SYSTEM BaggageSystemCTL (* System Configuration *)
  (* Standard: 61499-1 *)
  (* Version 0.3, 2003-12-05, JHC, Rockwell Automation, Renamed from NEWSYSTEM. *)
  (* Version 0.2, 2002-11-05, JHC, Rockwell Automation, Fixed missing (empty) FBD in Application. *)
  (* Version 0.1, 2002-01-17, JHC, Rockwell Automation, Minor cleanup *)
  (* Version 0.0, 2000-05-27, JHC, Rockwell Automation *)
  APPLICATION APP1
  END_APPLICATION
  DEVICE VIEW : ImageDev(Length := 820, Height := 900)
    RESOURCE RES : ImageResource
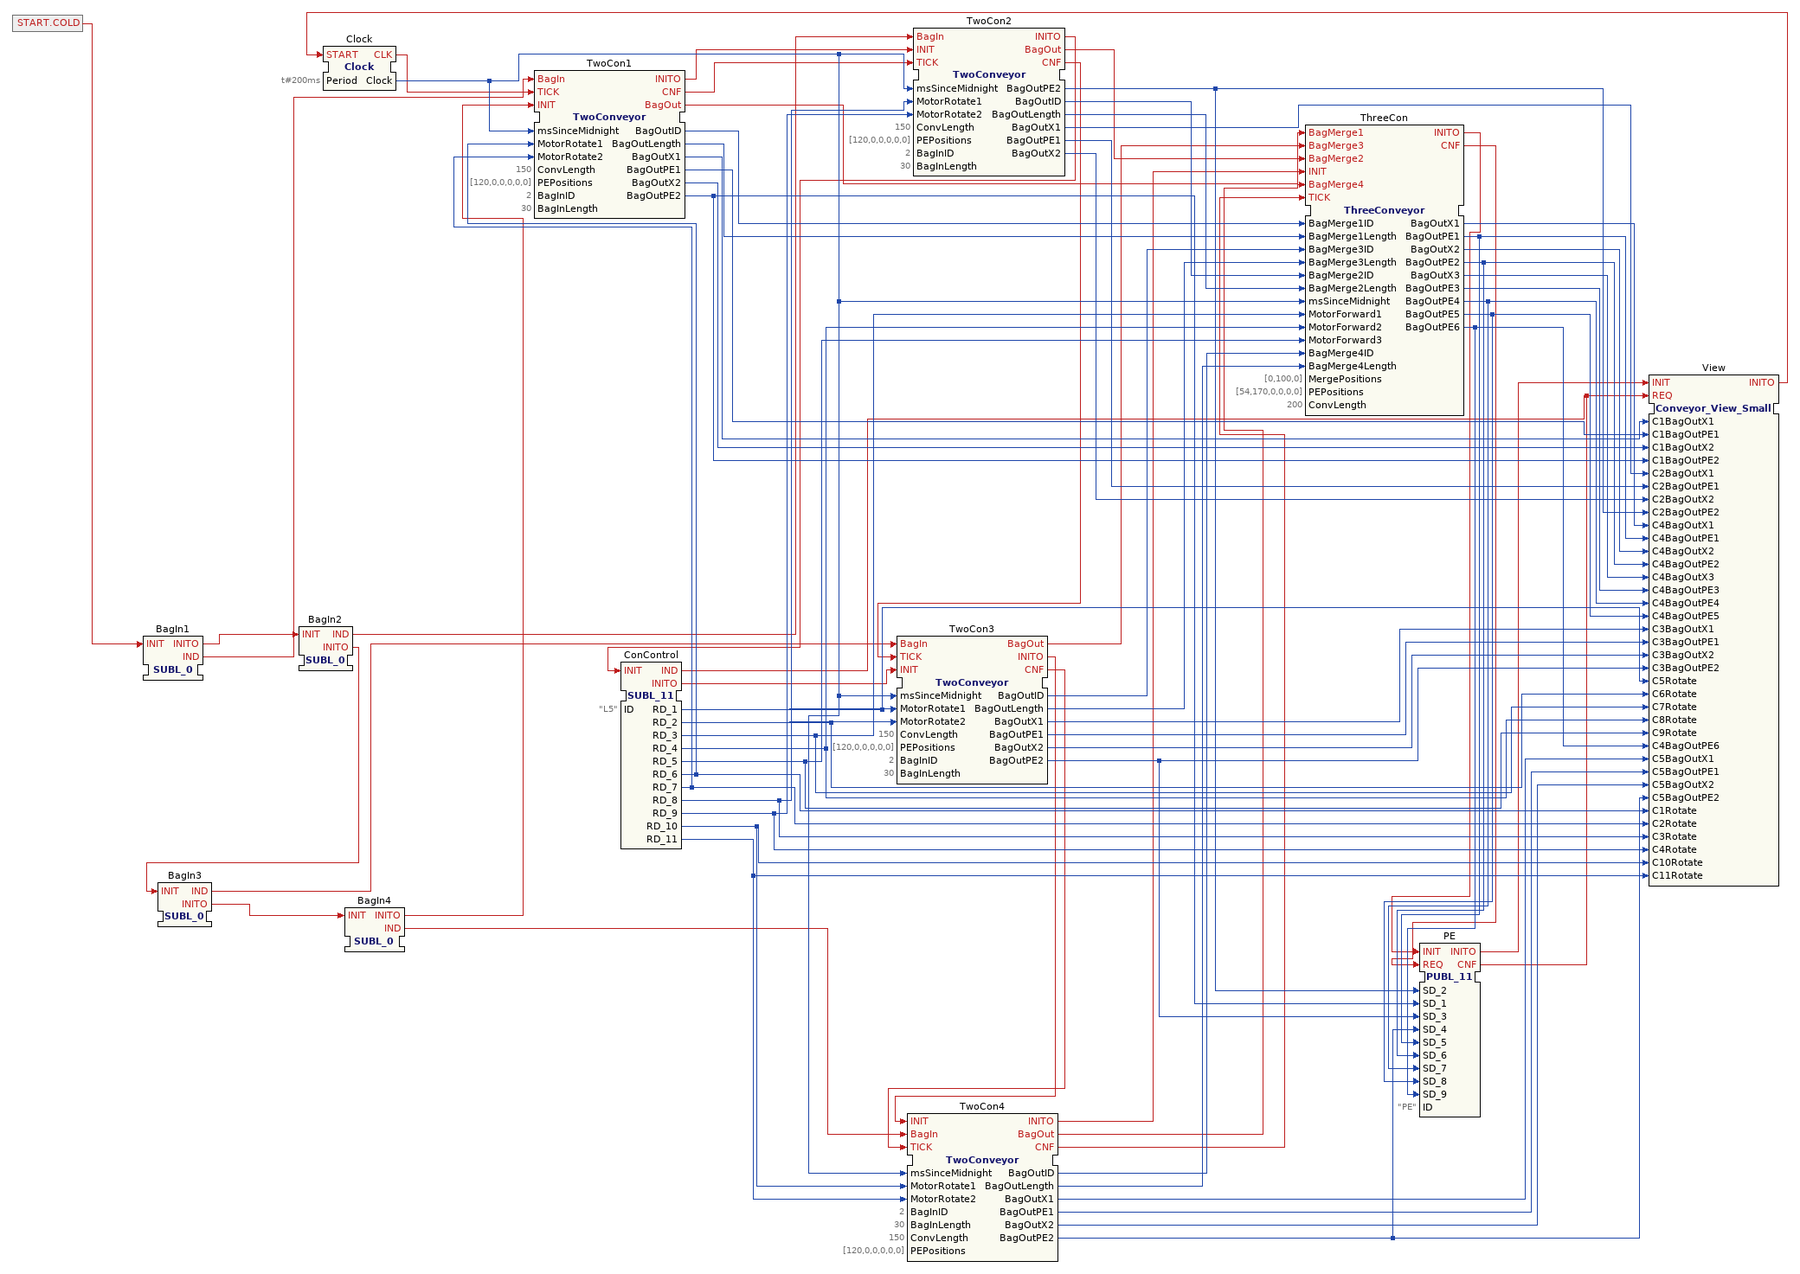
      FBS
        Clock : Clock(Period := t#200ms);
        View : Conveyor_View_Small;
        BagIn1 : SUBL_0;
        BagIn2 : SUBL_0;
        TwoCon1 : TwoConveyor(ConvLength := 150, PEPositions := [120,0,0,0,0,0], BagInID := 2, BagInLength := 30);
        TwoCon2 : TwoConveyor(ConvLength := 150, PEPositions := [120,0,0,0,0,0], BagInID := 2, BagInLength := 30);
        TwoCon3 : TwoConveyor(ConvLength := 150, PEPositions := [120,0,0,0,0,0], BagInID := 2, BagInLength := 30);
        ThreeCon : ThreeConveyor(MergePositions := [0,100,0], PEPositions := [54,170,0,0,0,0], ConvLength := 200);
        BagIn3 : SUBL_0;
        ConControl : SUBL_11(ID := "L5");
        PE : PUBL_11(ID := "PE");
        TwoCon4 : TwoConveyor(BagInID := 2, BagInLength := 30, ConvLength := 150, PEPositions := [120,0,0,0,0,0]);
        BagIn4 : SUBL_0;
      END_FBS
      EVENT_CONNECTIONS
        BagIn1.INITO TO BagIn2.INIT;
        BagIn1.IND TO TwoCon1.BagIn;
        BagIn2.IND TO TwoCon2.BagIn;
        BagIn3.IND TO TwoCon3.BagIn;
        TwoCon1.INITO TO TwoCon2.INIT;
        Clock.CLK TO TwoCon1.TICK;
        TwoCon1.CNF TO TwoCon2.TICK;
        TwoCon2.INITO TO ConControl.INIT;
        ThreeCon.INITO TO PE.INIT;
        ThreeCon.CNF TO PE.REQ;
        PE.INITO TO View.INIT;
        PE.CNF TO View.REQ;
        View.INITO TO Clock.START;
        TwoCon1.BagOut TO ThreeCon.BagMerge1;
        TwoCon3.BagOut TO ThreeCon.BagMerge3;
        TwoCon2.BagOut TO ThreeCon.BagMerge2;
        ConControl.IND TO View.REQ;
        TwoCon3.INITO TO TwoCon4.INIT;
        TwoCon4.INITO TO ThreeCon.INIT;
        TwoCon4.BagOut TO ThreeCon.BagMerge4;
        BagIn2.INITO TO BagIn3.INIT;
        BagIn3.INITO TO BagIn4.INIT;
        BagIn4.INITO TO TwoCon1.INIT;
        BagIn4.IND TO TwoCon4.BagIn;
        TwoCon2.CNF TO TwoCon3.TICK;
        TwoCon3.CNF TO TwoCon4.TICK;
        TwoCon4.CNF TO ThreeCon.TICK;
        ConControl.INITO TO TwoCon3.INIT;
        START.COLD TO BagIn1.INIT;
      END_CONNECTIONS
      DATA_CONNECTIONS
        TwoCon2.BagOutPE2 TO PE.SD_2;
        TwoCon1.BagOutID TO ThreeCon.BagMerge1ID;
        TwoCon1.BagOutLength TO ThreeCon.BagMerge1Length;
        TwoCon3.BagOutID TO ThreeCon.BagMerge3ID;
        TwoCon3.BagOutLength TO ThreeCon.BagMerge3Length;
        TwoCon2.BagOutID TO ThreeCon.BagMerge2ID;
        TwoCon2.BagOutLength TO ThreeCon.BagMerge2Length;
        Clock.Clock TO TwoCon1.msSinceMidnight;
        Clock.Clock TO TwoCon2.msSinceMidnight;
        Clock.Clock TO TwoCon3.msSinceMidnight;
        Clock.Clock TO ThreeCon.msSinceMidnight;
        TwoCon1.BagOutX1 TO View.C1BagOutX1;
        TwoCon1.BagOutPE1 TO View.C1BagOutPE1;
        TwoCon1.BagOutX2 TO View.C1BagOutX2;
        TwoCon1.BagOutPE2 TO View.C1BagOutPE2;
        TwoCon2.BagOutX1 TO View.C2BagOutX1;
        TwoCon2.BagOutPE1 TO View.C2BagOutPE1;
        TwoCon2.BagOutX2 TO View.C2BagOutX2;
        TwoCon2.BagOutPE2 TO View.C2BagOutPE2;
        ThreeCon.BagOutX1 TO View.C4BagOutX1;
        ThreeCon.BagOutPE1 TO View.C4BagOutPE1;
        ThreeCon.BagOutX2 TO View.C4BagOutX2;
        ThreeCon.BagOutPE2 TO View.C4BagOutPE2;
        ThreeCon.BagOutX3 TO View.C4BagOutX3;
        ThreeCon.BagOutPE3 TO View.C4BagOutPE3;
        ThreeCon.BagOutPE4 TO View.C4BagOutPE4;
        ThreeCon.BagOutPE5 TO View.C4BagOutPE5;
        TwoCon3.BagOutX1 TO View.C3BagOutX1;
        TwoCon3.BagOutPE1 TO View.C3BagOutPE1;
        TwoCon3.BagOutX2 TO View.C3BagOutX2;
        TwoCon3.BagOutPE2 TO View.C3BagOutPE2;
        ConControl.RD_1 TO TwoCon3.MotorRotate1;
        ConControl.RD_2 TO TwoCon3.MotorRotate2;
        ConControl.RD_3 TO ThreeCon.MotorForward1;
        ConControl.RD_4 TO ThreeCon.MotorForward2;
        ConControl.RD_5 TO ThreeCon.MotorForward3;
        TwoCon1.BagOutPE2 TO PE.SD_1;
        TwoCon3.BagOutPE2 TO PE.SD_3;
        ConControl.RD_1 TO View.C5Rotate;
        ConControl.RD_2 TO View.C6Rotate;
        ConControl.RD_3 TO View.C7Rotate;
        ConControl.RD_4 TO View.C8Rotate;
        ConControl.RD_5 TO View.C9Rotate;
        TwoCon4.BagOutID TO ThreeCon.BagMerge4ID;
        TwoCon4.BagOutLength TO ThreeCon.BagMerge4Length;
        ThreeCon.BagOutPE6 TO View.C4BagOutPE6;
        TwoCon4.BagOutX1 TO View.C5BagOutX1;
        TwoCon4.BagOutPE1 TO View.C5BagOutPE1;
        TwoCon4.BagOutX2 TO View.C5BagOutX2;
        TwoCon4.BagOutPE2 TO View.C5BagOutPE2;
        Clock.Clock TO TwoCon4.msSinceMidnight;
        ConControl.RD_6 TO TwoCon1.MotorRotate1;
        ConControl.RD_6 TO View.C1Rotate;
        ConControl.RD_7 TO TwoCon1.MotorRotate2;
        ConControl.RD_7 TO View.C2Rotate;
        ConControl.RD_8 TO TwoCon2.MotorRotate1;
        ConControl.RD_9 TO TwoCon2.MotorRotate2;
        ConControl.RD_8 TO View.C3Rotate;
        ConControl.RD_9 TO View.C4Rotate;
        ConControl.RD_10 TO TwoCon4.MotorRotate1;
        ConControl.RD_11 TO TwoCon4.MotorRotate2;
        ConControl.RD_10 TO View.C10Rotate;
        ConControl.RD_11 TO View.C11Rotate;
        TwoCon4.BagOutPE2 TO PE.SD_4;
        ThreeCon.BagOutPE1 TO PE.SD_5;
        ThreeCon.BagOutPE2 TO PE.SD_6;
        ThreeCon.BagOutPE4 TO PE.SD_7;
        ThreeCon.BagOutPE5 TO PE.SD_8;
        ThreeCon.BagOutPE6 TO PE.SD_9;
      END_CONNECTIONS
    END_RESOURCE
  END_DEVICE
  DEVICE HMI : FRAME_DEVICE(BOUNDS := [825,50,350,300], GRID := [1,6])
    RESOURCE RES1 : PANEL_RESOURCE
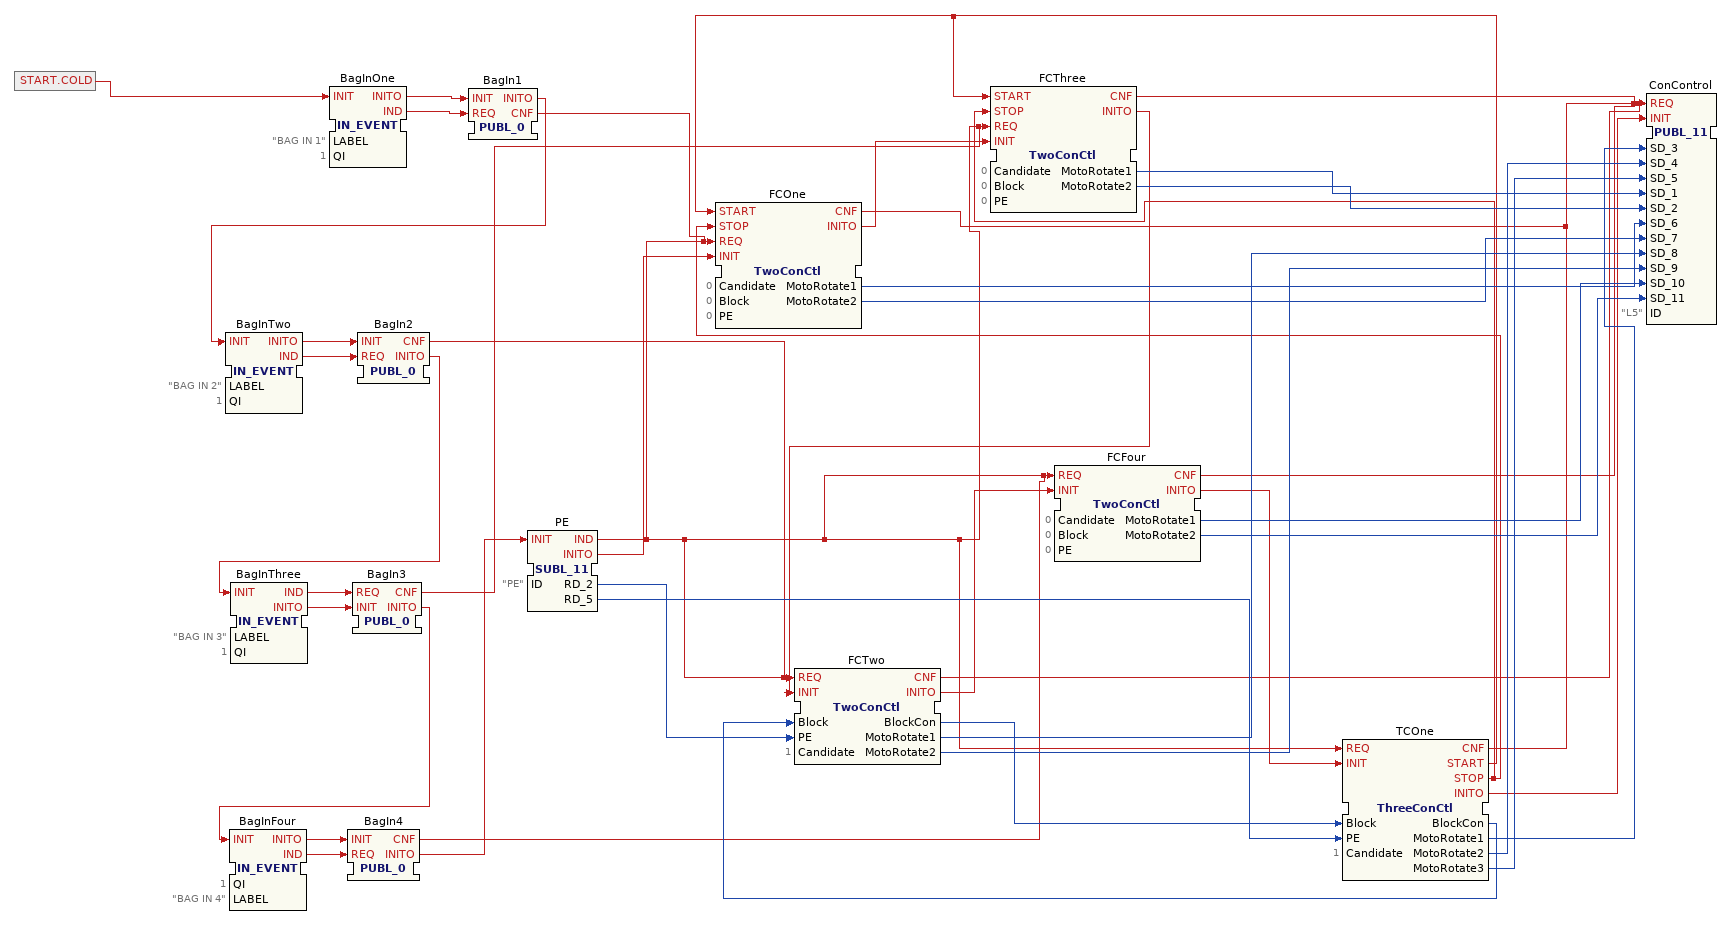
      FBS
        BagInOne : IN_EVENT(LABEL := "BAG IN 1", QI := 1);
        BagInThree : IN_EVENT(LABEL := "BAG IN 3", QI := 1);
        BagInTwo : IN_EVENT(LABEL := "BAG IN 2", QI := 1);
        BagIn1 : PUBL_0;
        BagIn3 : PUBL_0;
        BagIn2 : PUBL_0;
        FCOne : TwoConCtl(Candidate := 0, Block := 0, PE := 0);
        FCTwo : TwoConCtl(Candidate := 1);
        TCOne : ThreeConCtl(Candidate := 1);
        FCThree : TwoConCtl(Candidate := 0, Block := 0, PE := 0);
        ConControl : PUBL_11(ID := "L5");
        PE : SUBL_11(ID := "PE");
        BagInFour : IN_EVENT(QI := 1, LABEL := "BAG IN 4");
        BagIn4 : PUBL_0;
        FCFour : TwoConCtl(Candidate := 0, Block := 0, PE := 0);
      END_FBS
      EVENT_CONNECTIONS
        START.COLD TO BagInOne.INIT;
        BagInThree.IND TO BagIn3.REQ;
        BagInOne.INITO TO BagIn1.INIT;
        BagInOne.IND TO BagIn1.REQ;
        BagInThree.INITO TO BagIn3.INIT;
        BagIn1.INITO TO BagInTwo.INIT;
        BagInTwo.INITO TO BagIn2.INIT;
        PE.IND TO FCTwo.REQ;
        PE.IND TO TCOne.REQ;
        TCOne.CNF TO ConControl.REQ;
        FCThree.CNF TO ConControl.REQ;
        TCOne.START TO FCOne.START;
        TCOne.STOP TO FCOne.STOP;
        TCOne.START TO FCThree.START;
        TCOne.STOP TO FCThree.STOP;
        BagInTwo.IND TO BagIn2.REQ;
        PE.IND TO FCOne.REQ;
        PE.IND TO FCThree.REQ;
        BagIn1.CNF TO FCOne.REQ;
        BagIn2.CNF TO FCTwo.REQ;
        BagInFour.INITO TO BagIn4.INIT;
        PE.IND TO FCFour.REQ;
        BagInFour.IND TO BagIn4.REQ;
        BagIn4.CNF TO FCFour.REQ;
        BagIn3.CNF TO FCThree.REQ;
        FCOne.CNF TO ConControl.REQ;
        FCFour.CNF TO ConControl.REQ;
        FCTwo.CNF TO ConControl.REQ;
        BagIn2.INITO TO BagInThree.INIT;
        BagIn3.INITO TO BagInFour.INIT;
        BagIn4.INITO TO PE.INIT;
        PE.INITO TO FCOne.INIT;
        FCOne.INITO TO FCThree.INIT;
        FCThree.INITO TO FCTwo.INIT;
        FCTwo.INITO TO FCFour.INIT;
        FCFour.INITO TO TCOne.INIT;
        TCOne.INITO TO ConControl.INIT;
      END_CONNECTIONS
      DATA_CONNECTIONS
        FCTwo.BlockCon TO TCOne.Block;
        TCOne.BlockCon TO FCTwo.Block;
        TCOne.MotoRotate1 TO ConControl.SD_3;
        TCOne.MotoRotate2 TO ConControl.SD_4;
        TCOne.MotoRotate3 TO ConControl.SD_5;
        FCThree.MotoRotate1 TO ConControl.SD_1;
        FCThree.MotoRotate2 TO ConControl.SD_2;
        PE.RD_2 TO FCTwo.PE;
        FCOne.MotoRotate1 TO ConControl.SD_6;
        FCOne.MotoRotate2 TO ConControl.SD_7;
        FCTwo.MotoRotate1 TO ConControl.SD_8;
        FCTwo.MotoRotate2 TO ConControl.SD_9;
        FCFour.MotoRotate1 TO ConControl.SD_10;
        FCFour.MotoRotate2 TO ConControl.SD_11;
        PE.RD_5 TO TCOne.PE;
      END_CONNECTIONS
    END_RESOURCE
  END_DEVICE
END_SYSTEM
